Staubli VAL3: new.pgx

public program new(string x_sName (dimensions=1), num& x_nResult[] (dimensions=1))
  local num l_nResult
  local string l_sPrefix
begin
  // new one
  if save:nBoxType==1
    if insert(sml:box[x_sName])
      x_nResult=0
    else
      x_nResult=-1
    endIf
  elseIf save:nBoxType==2
    if insert(big:box[x_sName])
      x_nResult=0
    else
      x_nResult=-1
    endIf
  endIf
end
